
FUNCTION CB_bool_to_sint : INT


TITLE = ' Convert a boolean into an integer '
VERSION : '1.0'
AUTHOR  : CB
NAME    : boToSint
FAMILY  : TNI

VAR_INPUT
    IN : BOOL;
END_VAR

VAR_TEMP

END_VAR

BEGIN

CB_bool_to_sint := BOOL_TO_INT(IN);

END_FUNCTION
